// TIA Portal V20 export
// export: Created 2025-12-01T14:56:18.0505876Z, ExportSetting None, DisplayName Totally Integrated Automation Portal, DisplayVersion V20 Update 3, DisplayName TIA Portal Openness, DisplayVersion V20 Update 3, DisplayName TIA Portal Version Control Interface, DisplayVersion V20 Update 3, DisplayName STEP 7 Professional, DisplayVersion V20 Update 3, DisplayName STEP 7 Safety, DisplayVersion V20 Update 2, DisplayName WinCC Basic/Comfort/Advanced, DisplayVersion V20 Update 3, DisplayName WinCC Professional, DisplayVersion V20 Update 3, DisplayName WinCC Unified, DisplayVersion V20 Update 3
TYPE "UDT_HMI_SeñalesGalibo"
   STRUCT
      Alt_0_PaletVacio : Bool;
      Alt_1 : Bool;
      Alt_2 : Bool;
      Alt_3 : Bool;
      Alt_4 : Bool;
      Alt_Err : Bool;
      Anch_Der_1 : Bool;
      Anch_Der_2 : Bool;
      Anch_Der_3 : Bool;
      Anch_Der_Err : Bool;
      Anch_Izq_1 : Bool;
      Anch_Izq_2 : Bool;
      Anch_Izq_3 : Bool;
      Anch_Izq_Err : Bool;
      Front_1 : Bool;
      Front_2 : Bool;
      Front_3 : Bool;
      Hueco : Bool;
      HuecoRemon : Bool;
      Patin_1 : Bool;
      Patin_2 : Bool;
      Baliza : Bool;
      Frontal_Del_1 : Bool;
      Frontal_Del_2 : Bool;
      Frontal_Del_Err : Bool;
      Frontal_Tra_1 : Bool;
      Frontal_Tra_2 : Bool;
      Frontal_Tra_Err : Bool;
      Reserva_1 : Bool;
      Reserva_2 : Bool;
      Reserva_3 : Bool;
      Reserva_4 : Bool;
   END_STRUCT;
END_TYPE
